Yaskawa INFORM job: R1_W49-52-A2(90,90)KM-OK.JBI

/JOB
//NAME R1_W49-52-A2(90,90)KM-OK
///FOLDERNAME KRIS-SCIANA
//POS
///NPOS 60,60,0,3,0,0
///TOOL 0
///POSTYPE PULSE
///PULSE
C00000=67926,9987,-32186,8998,95712,36092
C00001=73499,59357,16168,-6018,120916,36656
C00002=82155,60075,23840,-4095,117096,40105
C00003=80395,50494,36025,-4582,109035,38821
C00004=80395,51517,40756,-4512,106656,38913
C00005=80395,52027,42770,-4486,105682,38950
C00006=80223,51226,42628,-4519,105350,38900
C00007=80395,52027,42770,-4486,105682,38950
C00008=80980,56111,48510,-6351,116206,43947
C00009=80818,54927,47183,-6433,116399,43872
C00010=81202,52432,43534,-5280,115457,44067
C00011=84530,48027,43385,-32270,97431,38822
C00012=83989,49026,44472,-32329,97091,38702
C00013=81922,49600,42415,-27580,98979,37293
C00014=80391,52535,44703,-25163,100687,36309
C00015=80390,52279,43783,-25205,101081,36222
C00016=120616,63440,59158,6431,95989,37803
C00017=120607,44118,38205,6262,90744,36049
C00018=120604,37989,32557,6266,87169,35869
C00019=120616,65158,62908,6289,94952,36261
C00020=120616,65746,64125,-3693,94481,36863
C00021=120616,64285,63377,-3690,94190,36871
C00022=120616,65746,64125,-3693,94481,36863
C00023=120616,64417,60871,-3703,95798,36824
C00024=120163,15436,13255,7554,71301,81964
C00025=120597,13122,10479,7433,71781,82150
C00026=120597,16200,13227,7437,71672,82143
C00027=120603,15446,13354,7456,71206,82115
C00028=120864,15455,13299,7392,71219,82211
C00029=121406,15306,13105,7263,71215,82403
C00030=120602,14724,11117,7415,72207,82177
C00031=120601,14277,6568,7325,74757,82332
C00032=119572,-9787,-22551,2150,106726,53581
C00033=120520,18911,14454,2479,119496,54181
C00034=120609,18986,16217,2501,118785,54201
C00035=120823,-17620,-23889,2281,103493,53962
C00036=120750,-19190,-25404,2273,103620,53940
C00037=120586,-17262,-17549,-5444,113084,56408
C00038=120586,-18193,-19569,-5507,113815,56379
C00039=120585,-18818,-23103,-5601,115662,56286
C00040=120548,-51762,-76595,-5198,106937,56689
C00041=85553,-40355,-70125,-3815,106956,45008
C00042=76137,-46433,-46321,45668,68230,62811
C00043=78373,-13498,-15012,50474,87103,54975
C00044=81252,9577,11862,53057,96291,49340
C00045=81044,37621,42001,55654,108833,42841
C00046=87827,57577,69560,49384,111543,37459
C00047=90576,58382,73628,49793,108703,37319
C00048=90743,51573,64806,49238,104953,51690
C00049=91111,57375,72470,50059,108548,37517
C00050=91309,60163,76105,49900,107913,37261
C00051=92072,49278,62084,49790,104576,52174
C00052=87096,38072,46331,51854,102603,47632
C00053=87827,57577,69560,49384,111543,37459
C00054=79802,34559,43026,59451,107818,42471
C00055=74570,40677,41733,59559,113121,43146
C00056=73532,31386,19668,63587,118165,46959
C00057=67438,12402,-14878,64444,108244,55096
C00058=37909,-135077,-127395,61795,76709,48061
C00059=1489,-133805,-127025,57463,40778,-58476
BC00000=261353,1145182,1068217
BC00001=261353,1145182,1068217
BC00002=261353,1145182,1068217
BC00003=261803,1145410,1068222
BC00004=263846,1148763,1068222
BC00005=264663,1150104,1068222
BC00006=264663,1150104,1068222
BC00007=264663,1150104,1068222
BC00008=273875,1134495,1046159
BC00009=273875,1134495,1046159
BC00010=273875,1134495,1046159
BC00011=227574,1140234,1046641
BC00012=227574,1140234,1046641
BC00013=227574,1140234,1046641
BC00014=225826,1138744,1053963
BC00015=221457,1135018,1068222
BC00016=383182,1191142,1068222
BC00017=382984,1191142,1068222
BC00018=382972,1191142,1068222
BC00019=382984,1191142,1068222
BC00020=365570,1191142,1068222
BC00021=365554,1191142,1068222
BC00022=365570,1191142,1068222
BC00023=365042,1191142,1068222
BC00024=395402,1191142,1068222
BC00025=398156,1191142,1068222
BC00026=398156,1191142,1068222
BC00027=395402,1191142,1068222
BC00028=393377,1191142,1068222
BC00029=390624,1191142,1068222
BC00030=391038,1191142,1068222
BC00031=392072,1191142,1068222
BC00032=378776,1124145,1068222
BC00033=381138,1126700,1068222
BC00034=382082,1127723,1068222
BC00035=382082,1127723,1068222
BC00036=382082,1127723,1068222
BC00037=373014,1102498,1068222
BC00038=371778,1100686,1068222
BC00039=368765,1096375,1068222
BC00040=368765,1096375,1068222
BC00041=368765,1096375,1068222
BC00042=395053,1169485,1068222
BC00043=395053,1169485,1068222
BC00044=395053,1169485,1068222
BC00045=395053,1169485,1068222
BC00046=395053,1169485,1068222
BC00047=395053,1169485,1068222
BC00048=395051,1170422,1068218
BC00049=395053,1170423,1068222
BC00050=395053,1170423,1068222
BC00051=395051,1170422,1068218
BC00052=395051,1170422,1068218
BC00053=395053,1169485,1068222
BC00054=395053,1169485,1068222
BC00055=395053,1169485,1068222
BC00056=395053,1169485,1068222
BC00057=395053,1169485,1068222
BC00058=395053,1188333,1068222
BC00059=96481,1188333,1068222
///POSTYPE BASE
///RECTAN
///RCONF 0,0,0,0,0,0,0,0,0,0,0,0,0,0,0,0,0,0,0,0,0,0,0,0
P00006=0.222,-3.123,-1.508,0.0000,0.0000,0.0000
P00023=0.143,-0.036,0.682,0.0000,0.0000,0.0000
P00024=0.145,-0.552,1.326,0.0000,0.0000,0.0000
//INST
///DATE 2024/07/24 16:17
///ATTR SC,RW
///GROUP1 RB1,BS1
NOP
'r1_W49-52-A2(90,90)(z_reki)
'Path S1175
SFTOF
MOVJ C00000 BC00000 VJ=100.00
MOVJ C00001 BC00001 VJ=100.00
MOVJ C00002 BC00002 VJ=100.00
MOVJ C00003 BC00003 VJ=15.00
MOVJ C00004 BC00004 VJ=10.00
MOVL C00005 BC00005 V=60.0
REFP 3 C00006 BC00006
CALL JOB:SEARCH-R1
SET P024 P006
SFTON P024
MOVL C00007 BC00007 V=60.0
MOVL C00008 BC00008 V=60.0
REFP 3 C00009 BC00009
CALL JOB:SEARCH-R1
SET P024 P006
SFTON P024
MOVL C00010 BC00010 V=60.0
MOVL C00011 BC00011 V=60.0
REFP 3 C00012 BC00012
CALL JOB:SEARCH-R1
SET P024 P006
SFTON P024
MOVL C00013 BC00013 V=100.0
MOVL C00014 BC00014 V=166.7
MOVL C00015 BC00015 V=250.0
'Path S1176
SFTOF
MOVL C00016 BC00016 V=250.0
MOVL C00017 BC00017 V=100.0
REFP 3 C00018 BC00018
CALL JOB:SEARCH-R1
SET P023 P006
SFTON P023
MOVL C00019 BC00019 V=133.3
MOVL C00020 BC00020 V=100.0
REFP 3 C00021 BC00021
CALL JOB:SEARCH-R1
SET P023 P006
SFTON P023
MOVL C00022 BC00022 V=60.0
SFTOF
MOVL C00023 BC00023 V=133.3
'Path W1177
SFTOF
SFTON P023
MOVL C00024 BC00024 V=200.0 PL=0
REFP 1 C00025 BC00025
REFP 2 C00026 BC00026
MACRO1 MJ#(0) ARGF7
ARCON
MOVL C00027 BC00027 V=10.8
MOVL C00028 BC00028 V=10.8
MOVL C00029 BC00029 V=10.8
ARCOF
MOVL C00030 BC00030 V=166.7
MOVL C00031 BC00031 V=166.7
SFTOF
'Path W1178
SFTOF
SFTON P024
MOVJ C00032 BC00032 VJ=15.00
MOVJ C00033 BC00033 VJ=15.00
MOVL C00034 BC00034 V=100.0 PL=0
REFP 1 C00035 BC00035
REFP 2 C00036 BC00036
MACRO1 MJ#(0) ARGF9
ARCON
MOVL C00037 BC00037 V=10.0
ARCOF
MOVL C00038 BC00038 V=100.0
MOVL C00039 BC00039 V=166.7
SFTOF
'Path VIA1213
SFTOF
MOVJ C00040 BC00040 VJ=20.00
'Path VIA1214
SFTOF
MOVJ C00041 BC00041 VJ=100.00
'Path VIA1222
SFTOF
MOVJ C00042 BC00042 VJ=15.00
'Path VIA1221
SFTOF
MOVJ C00043 BC00043 VJ=15.00
'Path VIA1220
SFTOF
MOVJ C00044 BC00044 VJ=10.00
MOVJ C00045 BC00045 VJ=10.00
'Path VIA1219
SFTOF
MOVJ C00046 BC00046 VJ=15.00
'Path W1179
SFTOF
SFTON P024
MOVJ C00047 BC00047 VJ=15.00
MOVL C00048 BC00048 V=100.0 PL=0
REFP 1 C00049 BC00049
REFP 2 C00050 BC00050
MACRO1 MJ#(0) ARGF0
MOVL C00051 BC00051 V=10.0
ARCOF
MOVL C00052 BC00052 V=166.7
SFTOF
'Path VIA1215
SFTOF
MOVJ C00053 BC00053 VJ=10.00
'Path VIA1216
SFTOF
MOVJ C00054 BC00054 VJ=10.00
'Path VIA1217
SFTOF
MOVJ C00055 BC00055 VJ=15.00
'Path VIA1218
SFTOF
MOVJ C00056 BC00056 VJ=15.00
MOVJ C00057 BC00057 VJ=100.00
MOVJ C00058 BC00058 VJ=100.00
MOVJ C00059 BC00059 VJ=100.00
END
